(* IEC 61131-3 sources: crb-codesys/generation/scripts/repoeval/重型运输系统/core/PRG, 12 files *)

(* ---- Barrier.st ---- *)
PROGRAM Barrier
VAR
	bInit			:BOOL:=TRUE;
	initCount		:INT:= 100 * 2;		//2s后开始初始化，执行
	timeout			:INT:= 100 * 16;	//10ms间隔时 is 15 second
	timeexe			:INT:= 100 * 8;		//需要停止时，额外执行指令时间
	cmdExecutor0	:CommandExecutor0;
	cmdExecutor		:CommandExecutor;
	grdPid			:ARRAY[1..10] OF grdPosCtrl;
	skyPid			:ARRAY[0..10] OF skyPosCtrl;
	resetPidParam	:BOOL;							//pid参数复位
	pidMode			:BOOL;							//使用pid控制
	autoButtonMode	:BOOL;							//手动复位按钮
	autoEnableMode	:BOOL;							//有动作时使能自动开启
	autoPctMode		:BOOL;
	manualPidPrmSet	:BOOL;							//manualPidParamSet,手动设定pid位置参数

	gi				:INT;			//ground-i
	si				:INT;			//sky-i

	level			:INT;			//1->地轨	2->天轨
	idx				:INT := -1 ;	//挡板索引编号
END_VAR

//初始化
IF initCount = 0 THEN
	IF bInit THEN
		initialize();
		initializePid();
		bInit := FALSE;
	END_IF
ELSE
	initCount := initCount - 1;
	RETURN;
END_IF

//指令执行
pidTestUi();

IF pidMode THEN
	pidCalc();
	pidExecute();
ELSE
	IF autoPctMode THEN setExecutePercent(); END_IF
	manualExecute();
END_IF

//界面交互
interfaceAct();

//状态更新
updateStatus(error := 1);

//复位按钮模式/
IF autoButtonMode THEN
	autoResetButton();
END_IF
IF autoEnableMode THEN
	autoEnable();
END_IF

(* ---- Barrier_autoEnable.st ---- *)
IF pidMode THEN 	//pid模式，没有动作指令时不执行输出

	IF NOT manualPidPrmSet THEN
		FOR gi := 1 TO 10 DO
			 IF gDev.grd[gi].vector = TargetDirect.stop THEN
				cmdExecutor(level := 1, idx := gi, percent := 0);
			 END_IF
		END_FOR

		FOR si := 1 TO 10 DO
			IF gDev.sky[si].vector = TargetDirect.stop THEN
				cmdExecutor(level := 2, idx := si, percent := 0);
			END_IF
		END_FOR
		//起竖挡板执行开关量特判
		IF gDev.sky[0].vector = TargetDirect.stop THEN
			cmdExecutor(level := 2, idx := 0, percent := 0);
		END_IF
	END_IF
ELSE		//开关量控制

	FOR gi := 1 TO 10 DO
		 IF gDev.grd[gi].vector = TargetDirect.stop THEN
			gUI.grd[gi].pwrEnable := FALSE;
		 ELSE
			gUI.grd[gi].pwrEnable := TRUE;
		 END_IF
	END_FOR

	FOR si := 0 TO 10 DO
		IF gDev.sky[si].vector = TargetDirect.stop THEN
			gUI.sky[si].pwrEnable := FALSE;
		ELSE
			gUI.sky[si].pwrEnable := TRUE;
		END_IF
	END_FOR
END_IF

(*
FOR gi := 1 TO 10 DO
	 IF gDev.grd[gi].vector <> TargetDirect.stop THEN
		IF pidMode THEN
			cmdExecutor(level := 1, idx := gi, percent := grdPid[gi].res);
		ELSE
			gUI.grd[gi].pwrEnable := TRUE;
		END_IF
	 ELSE
		IF pidMode THEN
			cmdExecutor(level := 1, idx := gi, percent := 0);
		ELSE
			gUI.grd[gi].pwrEnable := FALSE;
		END_IF
	 END_IF
END_FOR

FOR si := 1 TO 10 DO
	IF gDev.sky[si].vector <> TargetDirect.stop THEN		//运动状态，执行  PID或开关使能
		IF pidMode THEN
			cmdExecutor(level := 2, idx := si, percent := skyPid[si].res);
		ELSE
			gUI.sky[si].pwrEnable := TRUE;
		END_IF
	ELSE													//停止状态，关闭 PID或开关使能
		IF pidMode THEN
			cmdExecutor(level := 2, idx := si, percent := 0);
		ELSE
			gUI.sky[si].pwrEnable := FALSE;
		END_IF
	END_IF
END_FOR

IF gDev.sky[0].vector <> TargetDirect.stop THEN
	gUI.sky[0].pwrEnable := TRUE;
	IF gDev.sky[0].vector = TargetDirect.extend THEN	cmdExecutor(level := 2, idx := 0, percent := gDev.sky[0].ctrl.exPct);END_IF
	IF gDev.sky[0].vector = TargetDirect.retract THEN	cmdExecutor(level := 2, idx := 0, percent := -gDev.sky[0].ctrl.rtPct);END_IF
ELSE
	gUI.sky[0].pwrEnable := FALSE;
	cmdExecutor(level := 2, idx := 0, percent := 0);
END_IF
*)

(* ---- Barrier_autoReseButton.st ---- *)
//更新Button
FOR gi := 1 TO 10 DO
	setButtonByDirect(1, gi, gDev.grd[gi].vector);
END_FOR

FOR si := 0 TO 10 DO
	setButtonByDirect(2, si, gDev.sky[si].vector);
END_FOR

(* ---- Barrier_initialize.st ---- *)
//默认自动使能
gUI.mode.autoEnable	:= TRUE;
gUI.mode.usePID := TRUE;

//initialize boundary val
	//ground
	gDev.grd[	1	].sensor.retractVal	:=	4.4	;		gDev.grd[	1	].sensor.extendVal	:=	108 	;
	gDev.grd[	2	].sensor.retractVal	:=	3.5	;		gDev.grd[	2	].sensor.extendVal	:=	113.4	;
	gDev.grd[	3	].sensor.retractVal	:=	4.1	;		gDev.grd[	3	].sensor.extendVal	:=	110 	;
	gDev.grd[	4	].sensor.retractVal	:=	1	;		gDev.grd[	4	].sensor.extendVal	:=	112.3	;		//结构问题暂不动
	gDev.grd[	5	].sensor.retractVal	:=	4.0	;		gDev.grd[	5	].sensor.extendVal	:=	107.1-0.5	;
	gDev.grd[	6	].sensor.retractVal	:=	3.5	;		gDev.grd[	6	].sensor.extendVal	:=	110.5	;
	gDev.grd[	7	].sensor.retractVal	:=	5	;		gDev.grd[	7	].sensor.extendVal	:=	109.7   ;
	gDev.grd[	8	].sensor.retractVal	:=	4.8	;		gDev.grd[	8	].sensor.extendVal	:=	109.2	;
	gDev.grd[	9	].sensor.retractVal	:=	3.2	;		gDev.grd[	9	].sensor.extendVal	:=	108 -0.5 	;
	gDev.grd[	10	].sensor.retractVal	:=	6.9	;		gDev.grd[	10	].sensor.extendVal	:=	112 	;
(*
	gDev.grd[	7	].sensor.retractVal	:=	3.6	;		gDev.grd[	7	].sensor.extendVal	:=	108.3	;
	gDev.grd[	8	].sensor.retractVal	:=	3.5	;		gDev.grd[	8	].sensor.extendVal	:=	113.1	;
	gDev.grd[	9	].sensor.retractVal	:=	3.2	;		gDev.grd[	9	].sensor.extendVal	:=	107.3	;
	gDev.grd[	10	].sensor.retractVal	:=	3.4	;		gDev.grd[	10	].sensor.extendVal	:=	113.5	;*)

	//sky
	gDev.sky[	0	].sensor.retractVal	:=	3.7	;		gDev.sky[	0	].sensor.extendVal	:=	213.6	;
	gDev.sky[	1	].sensor.retractVal	:=	8.8	;		gDev.sky[	1	].sensor.extendVal	:=	113.1	;
	gDev.sky[	2	].sensor.retractVal	:=	3.5	;		gDev.sky[	2	].sensor.extendVal	:=	113.0	;
	gDev.sky[	3	].sensor.retractVal	:=	3.5	;		gDev.sky[	3	].sensor.extendVal	:=	111.0	;
	gDev.sky[	4	].sensor.retractVal	:=	1	;		gDev.sky[	4	].sensor.extendVal	:=	58.2	;
	gDev.sky[	5	].sensor.retractVal	:=	3.2	;		gDev.sky[	5	].sensor.extendVal	:=	106.6	;
	gDev.sky[	6	].sensor.retractVal	:=	6.2	;		gDev.sky[	6	].sensor.extendVal	:=	109.8	;
(*
	gDev.sky[	7	].sensor.retractVal	:=	1	;		gDev.sky[	7	].sensor.extendVal	:=	113.4	;		//default:115
	gDev.sky[	8	].sensor.retractVal	:=	1	;		gDev.sky[	8	].sensor.extendVal	:=	112.2	;
	gDev.sky[	9	].sensor.retractVal	:=	1	;		gDev.sky[	9	].sensor.extendVal	:=	112.3	;
	gDev.sky[	10	].sensor.retractVal	:=	1	;		gDev.sky[	10	].sensor.extendVal	:=	66.3	;
*)

	gDev.sky[	7	].sensor.retractVal	:=	5	;		gDev.sky[	7	].sensor.extendVal	:=	108.7	;		//default:115
	gDev.sky[	8	].sensor.retractVal	:=	8.6	;		gDev.sky[	8	].sensor.extendVal	:=	113.3	;
	gDev.sky[	9	].sensor.retractVal	:=	12.9 ;		gDev.sky[	9	].sensor.extendVal	:=	113.8	;
	gDev.sky[	10	].sensor.retractVal	:=	3.9 ;		gDev.sky[	10	].sensor.extendVal	:=	111.5	;

//初始化默认伸缩比例量
	gDev.grd[1].ctrl.exPct :=	28		;			gDev.grd[1].ctrl.rtPct :=	25		;
	gDev.grd[2].ctrl.exPct :=	28		;			gDev.grd[2].ctrl.rtPct :=	25		;
	gDev.grd[3].ctrl.exPct :=	30		;			gDev.grd[3].ctrl.rtPct :=	25		;
	gDev.grd[4].ctrl.exPct :=	28		;			gDev.grd[4].ctrl.rtPct :=	25		;
	gDev.grd[5].ctrl.exPct :=	33		;			gDev.grd[5].ctrl.rtPct :=	33		;		//exPct:=26	rtPct:=21 二次比例
	gDev.grd[6].ctrl.exPct :=	28		;			gDev.grd[6].ctrl.rtPct :=	25		;
	gDev.grd[7].ctrl.exPct :=	28		;			gDev.grd[7].ctrl.rtPct :=	25		;
	gDev.grd[8].ctrl.exPct :=	28		;			gDev.grd[8].ctrl.rtPct :=	25		;
	gDev.grd[9].ctrl.exPct :=	28		;			gDev.grd[9].ctrl.rtPct :=	25		;
	gDev.grd[10].ctrl.exPct :=	28		;			gDev.grd[10].ctrl.rtPct :=	25		;

	gDev.sky[0].ctrl.exPct :=	35		;			gDev.sky[0].ctrl.rtPct :=	41		;
	gDev.sky[1].ctrl.exPct :=	25		;			gDev.sky[1].ctrl.rtPct :=	28		;
	gDev.sky[2].ctrl.exPct :=	25		;			gDev.sky[2].ctrl.rtPct :=	28		;
	gDev.sky[3].ctrl.exPct :=	25		;			gDev.sky[3].ctrl.rtPct :=	28		;
	gDev.sky[4].ctrl.exPct :=	25		;			gDev.sky[4].ctrl.rtPct :=	28		;
	gDev.sky[5].ctrl.exPct :=	27		;			gDev.sky[5].ctrl.rtPct :=	30.5	;
	gDev.sky[6].ctrl.exPct :=	25		;			gDev.sky[6].ctrl.rtPct :=	29		;
	gDev.sky[7].ctrl.exPct :=	25		;			gDev.sky[7].ctrl.rtPct :=	28		;
	gDev.sky[8].ctrl.exPct :=	25		;			gDev.sky[8].ctrl.rtPct :=	28		;
	gDev.sky[9].ctrl.exPct :=	25		;			gDev.sky[9].ctrl.rtPct :=	28		;
	gDev.sky[10].ctrl.exPct :=	25		;			gDev.sky[10].ctrl.rtPct :=	28		;

//initialize device name

											gUI.sky[	0	].wname	:=	"天轨1#"	;
gUI.grd[	1	].wname	:=	"地轨1#"	;	gUI.sky[	1	].wname	:=	"天轨2#"	;
gUI.grd[	2	].wname	:=	"地轨2#"	;	gUI.sky[	2	].wname	:=	"天轨3#"	;
gUI.grd[	3	].wname	:=	"地轨3#"	;	gUI.sky[	3	].wname	:=	"天轨4#"	;
gUI.grd[	4	].wname	:=	"地轨4#"	;	gUI.sky[	4	].wname	:=	"天轨5#"	;
gUI.grd[	5	].wname	:=	"地轨5#"	;	gUI.sky[	5	].wname	:=	"天轨6#"	;
gUI.grd[	6	].wname	:=	"地轨6#"	;	gUI.sky[	6	].wname	:=	"天轨7#"	;
gUI.grd[	7	].wname	:=	"地轨7#"	;	gUI.sky[	7	].wname	:=	"天轨8#"	;
gUI.grd[	8	].wname	:=	"地轨8#"	;	gUI.sky[	8	].wname	:=	"天轨9#"	;
gUI.grd[	9	].wname	:=	"地轨9#"	;	gUI.sky[	9	].wname	:=	"天轨10#"	;
gUI.grd[	10	].wname	:=	"地轨10#"	;	gUI.sky[	10	].wname	:=	"天轨11#"	;

												gUI.sky[	0	].hzname	:=	"天.起竖"	;
gUI.grd[	1	].hzname	:=	"地.横1"	;	gUI.sky[	1	].hzname	:=	"天.横1"	;
gUI.grd[	2	].hzname	:=	"地.纵1"	;	gUI.sky[	2	].hzname	:=	"天.纵1"	;
gUI.grd[	3	].hzname	:=	"地.横2"	;	gUI.sky[	3	].hzname	:=	"天.横2"	;
gUI.grd[	4	].hzname	:=	"地.横3"	;	gUI.sky[	4	].hzname	:=	"天.横3"	;
gUI.grd[	5	].hzname	:=	"地.横4"	;	gUI.sky[	5	].hzname	:=	"天.横4"	;
gUI.grd[	6	].hzname	:=	"地.横5"	;	gUI.sky[	6	].hzname	:=	"天.横5"	;
gUI.grd[	7	].hzname	:=	"地.纵2"	;	gUI.sky[	7	].hzname	:=	"天.纵2"	;
gUI.grd[	8	].hzname	:=	"地.横6"	;	gUI.sky[	8	].hzname	:=	"天.横6"	;
gUI.grd[	9	].hzname	:=	"地.横7"	;	gUI.sky[	9	].hzname	:=	"天.横7"	;
gUI.grd[	10	].hzname	:=	"地.横8"	;	gUI.sky[	10	].hzname	:=	"天.横8"	;

											gUI.sky[	0	].name	:=	'SKY_00'	;
gUI.grd[	1	].name	:=	'GRD_01'	;	gUI.sky[	1	].name	:=	'SKY_01'	;
gUI.grd[	2	].name	:=	'GRD_02'	;	gUI.sky[	2	].name	:=	'SKY_02'	;
gUI.grd[	3	].name	:=	'GRD_03'	;	gUI.sky[	3	].name	:=	'SKY_03'	;
gUI.grd[	4	].name	:=	'GRD_04'	;	gUI.sky[	4	].name	:=	'SKY_04'	;
gUI.grd[	5	].name	:=	'GRD_05'	;	gUI.sky[	5	].name	:=	'SKY_05'	;
gUI.grd[	6	].name	:=	'GRD_06'	;	gUI.sky[	6	].name	:=	'SKY_06'	;
gUI.grd[	7	].name	:=	'GRD_07'	;	gUI.sky[	7	].name	:=	'SKY_07'	;
gUI.grd[	8	].name	:=	'GRD_08'	;	gUI.sky[	8	].name	:=	'SKY_08'	;
gUI.grd[	9	].name	:=	'GRD_09'	;	gUI.sky[	9	].name	:=	'SKY_09'	;
gUI.grd[	10	].name	:=	'GRD_10'	;	gUI.sky[	10	].name	:=	'SKY_10'	;

//使用传感器当前位置作为初始化目标位移点
//(*
FOR gi := 1 TO 10 DO
	IF gDev.grd[gi].sensor.position <> 0.0 THEN
		gDev.grd[gi].ctrl.pos.Set_Point := gDev.grd[gi].sensor.position;
	ELSE
		gDev.grd[gi].ctrl.isError := TRUE;
	END_IF
END_FOR

FOR si := 0 TO 10 DO
	IF gDev.sky[si].sensor.position <> 0.0 THEN
		gDev.sky[si].ctrl.pos.Set_Point := gDev.sky[si].sensor.position;
	ELSE
		gDev.sky[si].ctrl.isError := TRUE;
	END_IF
END_FOR
//*)

(* ---- Barrier_initializePid.st ---- *)
//PID param
gDev.grd[	1	].ctrl.pos.Kp	:=	1.2	;	gDev.grd[	1	].ctrl.spd.Kp	:=	0.05	;
gDev.grd[	1	].ctrl.pos.Ki	:=	0	;	gDev.grd[	1	].ctrl.spd.Ki	:=	0		;
gDev.grd[	1	].ctrl.pos.Kd	:=	0	;	gDev.grd[	1	].ctrl.spd.Kd	:=	0.02	;

gDev.grd[	2	].ctrl.pos.Kp	:=	1.3	;	gDev.grd[	2	].ctrl.spd.Kp	:=	0.05	;
gDev.grd[	2	].ctrl.pos.Ki	:=	0	;	gDev.grd[	2	].ctrl.spd.Ki	:=	0		;
gDev.grd[	2	].ctrl.pos.Kd	:=	0	;	gDev.grd[	2	].ctrl.spd.Kd	:=	0.002	;
gDev.grd[	3	].ctrl.pos.Kp	:=	1	;	gDev.grd[	3	].ctrl.spd.Kp	:=	0.01	;
gDev.grd[	3	].ctrl.pos.Ki	:=	0	;	gDev.grd[	3	].ctrl.spd.Ki	:=	0		;
gDev.grd[	3	].ctrl.pos.Kd	:=	0	;	gDev.grd[	3	].ctrl.spd.Kd	:=	0		;

gDev.grd[	4	].ctrl.pos.Kp	:=	0	;	gDev.grd[	4	].ctrl.spd.Kp	:=	0		;
gDev.grd[	4	].ctrl.pos.Ki	:=	0	;	gDev.grd[	4	].ctrl.spd.Ki	:=	0		;
gDev.grd[	4	].ctrl.pos.Kd	:=	0	;	gDev.grd[	4	].ctrl.spd.Kd	:=	0		;
gDev.grd[	5	].ctrl.pos.Kp	:=	1.2	;	gDev.grd[	5	].ctrl.spd.Kp	:=	0.01	;
gDev.grd[	5	].ctrl.pos.Ki	:=	0	;	gDev.grd[	5	].ctrl.spd.Ki	:=	0		;
gDev.grd[	5	].ctrl.pos.Kd	:=	0	;	gDev.grd[	5	].ctrl.spd.Kd	:=	0		;

gDev.grd[	6	].ctrl.pos.Kp	:=	1.2	;	gDev.grd[	6	].ctrl.spd.Kp	:=	0.01	;
gDev.grd[	6	].ctrl.pos.Ki	:=	0	;	gDev.grd[	6	].ctrl.spd.Ki	:=	0		;
gDev.grd[	6	].ctrl.pos.Kd	:=	0	;	gDev.grd[	6	].ctrl.spd.Kd	:=	0		;
gDev.grd[	7	].ctrl.pos.Kp	:=	1.1	;	gDev.grd[	7	].ctrl.spd.Kp	:=	0.02		;
gDev.grd[	7	].ctrl.pos.Ki	:=	0	;	gDev.grd[	7	].ctrl.spd.Ki	:=	0		;
gDev.grd[	7	].ctrl.pos.Kd	:=	0	;	gDev.grd[	7	].ctrl.spd.Kd	:=	0		;

gDev.grd[	8	].ctrl.pos.Kp	:=	1.1	;	gDev.grd[	8	].ctrl.spd.Kp	:=	0.01		;
gDev.grd[	8	].ctrl.pos.Ki	:=	0	;	gDev.grd[	8	].ctrl.spd.Ki	:=	0		;
gDev.grd[	8	].ctrl.pos.Kd	:=	0	;	gDev.grd[	8	].ctrl.spd.Kd	:=	0		;
gDev.grd[	9	].ctrl.pos.Kp	:=	1.1	;	gDev.grd[	9	].ctrl.spd.Kp	:=	0.05		;
gDev.grd[	9	].ctrl.pos.Ki	:=	0	;	gDev.grd[	9	].ctrl.spd.Ki	:=	0		;
gDev.grd[	9	].ctrl.pos.Kd	:=	0	;	gDev.grd[	9	].ctrl.spd.Kd	:=	0		;
gDev.grd[	10	].ctrl.pos.Kp	:=	1.1	;	gDev.grd[	10	].ctrl.spd.Kp	:=	0.02		;
gDev.grd[	10	].ctrl.pos.Ki	:=	0	;	gDev.grd[	10	].ctrl.spd.Ki	:=	0		;
gDev.grd[	10	].ctrl.pos.Kd	:=	0	;	gDev.grd[	10	].ctrl.spd.Kd	:=	0		;

gDev.sky[	0	].ctrl.pos.Kp	:=	1.0	;	gDev.sky[	0	].ctrl.spd.Kp	:=	0.01	;
gDev.sky[	0	].ctrl.pos.Ki	:=	0	;	gDev.sky[	0	].ctrl.spd.Ki	:=	0		;
gDev.sky[	0	].ctrl.pos.Kd	:=	0.1	;	gDev.sky[	0	].ctrl.spd.Kd	:=	0.001	;
gDev.sky[	1	].ctrl.pos.Kp	:=	1.0	;	gDev.sky[	1	].ctrl.spd.Kp	:=	0.01	;
gDev.sky[	1	].ctrl.pos.Ki	:=	0	;	gDev.sky[	1	].ctrl.spd.Ki	:=	0		;
gDev.sky[	1	].ctrl.pos.Kd	:=	0	;	gDev.sky[	1	].ctrl.spd.Kd	:=	0.001	;

gDev.sky[	2	].ctrl.pos.Kp	:=	1.1	;	gDev.sky[	2	].ctrl.spd.Kp	:=	0.02	;
gDev.sky[	2	].ctrl.pos.Ki	:=	0	;	gDev.sky[	2	].ctrl.spd.Ki	:=	0		;
gDev.sky[	2	].ctrl.pos.Kd	:=	0	;	gDev.sky[	2	].ctrl.spd.Kd	:=	0.001	;
gDev.sky[	3	].ctrl.pos.Kp	:=	1.1	;	gDev.sky[	3	].ctrl.spd.Kp	:=	0.02	;
gDev.sky[	3	].ctrl.pos.Ki	:=	0	;	gDev.sky[	3	].ctrl.spd.Ki	:=	0		;
gDev.sky[	3	].ctrl.pos.Kd	:=	0.02;	gDev.sky[	3	].ctrl.spd.Kd	:=	0.001	;

gDev.sky[	4	].ctrl.pos.Kp	:=	0	;	gDev.sky[	4	].ctrl.spd.Kp	:=	0		;
gDev.sky[	4	].ctrl.pos.Ki	:=	0	;	gDev.sky[	4	].ctrl.spd.Ki	:=	0		;
gDev.sky[	4	].ctrl.pos.Kd	:=	0	;	gDev.sky[	4	].ctrl.spd.Kd	:=	0		;
gDev.sky[	5	].ctrl.pos.Kp	:=	1.2	;	gDev.sky[	5	].ctrl.spd.Kp	:=	0.01	;
gDev.sky[	5	].ctrl.pos.Ki	:=	0	;	gDev.sky[	5	].ctrl.spd.Ki	:=	0		;
gDev.sky[	5	].ctrl.pos.Kd	:=	0	;	gDev.sky[	5	].ctrl.spd.Kd	:=	0.001	;

gDev.sky[	6	].ctrl.pos.Kp	:=	1.1	;	gDev.sky[	6	].ctrl.spd.Kp	:=	0.01	;
gDev.sky[	6	].ctrl.pos.Ki	:=	0	;	gDev.sky[	6	].ctrl.spd.Ki	:=	0		;
gDev.sky[	6	].ctrl.pos.Kd	:=	0.01;	gDev.sky[	6	].ctrl.spd.Kd	:=	0.001	;
gDev.sky[	7	].ctrl.pos.Kp	:=	1.1	;	gDev.sky[	7	].ctrl.spd.Kp	:=	0.01	;
gDev.sky[	7	].ctrl.pos.Ki	:=	0	;	gDev.sky[	7	].ctrl.spd.Ki	:=	0		;
gDev.sky[	7	].ctrl.pos.Kd	:=	0	;	gDev.sky[	7	].ctrl.spd.Kd	:=	0		;

gDev.sky[	8	].ctrl.pos.Kp	:=	1.1	;	gDev.sky[	8	].ctrl.spd.Kp	:=	0.01	;
gDev.sky[	8	].ctrl.pos.Ki	:=	0	;	gDev.sky[	8	].ctrl.spd.Ki	:=	0		;
gDev.sky[	8	].ctrl.pos.Kd	:=	0	;	gDev.sky[	8	].ctrl.spd.Kd	:=	0		;
gDev.sky[	9	].ctrl.pos.Kp	:=	1.2	;	gDev.sky[	9	].ctrl.spd.Kp	:=	0.01		;
gDev.sky[	9	].ctrl.pos.Ki	:=	0	;	gDev.sky[	9	].ctrl.spd.Ki	:=	0		;
gDev.sky[	9	].ctrl.pos.Kd	:=	0	;	gDev.sky[	9	].ctrl.spd.Kd	:=	0		;
gDev.sky[	10	].ctrl.pos.Kp	:=	1.1	;	gDev.sky[	10	].ctrl.spd.Kp	:=	0		;
gDev.sky[	10	].ctrl.pos.Ki	:=	0	;	gDev.sky[	10	].ctrl.spd.Ki	:=	0		;
gDev.sky[	10	].ctrl.pos.Kd	:=	0	;	gDev.sky[	10	].ctrl.spd.Kd	:=	0		;

gDev.grd[1	].ctrl.ff.pstThreshold	:=	18.5	;	gDev.grd[1	].ctrl.ff.pstKv	:=	0.35 	;
gDev.grd[1	].ctrl.ff.negThreshold	:=	15  	;	gDev.grd[1	].ctrl.ff.negKv	:=	0.27	;
gDev.grd[2	].ctrl.ff.pstThreshold	:=	18  	;	gDev.grd[2	].ctrl.ff.pstKv	:=	0.27	;
gDev.grd[2	].ctrl.ff.negThreshold	:=	16  	;	gDev.grd[2	].ctrl.ff.negKv	:=	0.27	;
gDev.grd[3	].ctrl.ff.pstThreshold	:=	19  	;	gDev.grd[3	].ctrl.ff.pstKv	:=	0.3 	;
gDev.grd[3	].ctrl.ff.negThreshold	:=	16  	;	gDev.grd[3	].ctrl.ff.negKv	:=	0.3 	;
gDev.grd[4	].ctrl.ff.pstThreshold	:=	0   	;	gDev.grd[4	].ctrl.ff.pstKv	:=	0   	;
gDev.grd[4	].ctrl.ff.negThreshold	:=	0   	;	gDev.grd[4	].ctrl.ff.negKv	:=	0   	;
gDev.grd[5	].ctrl.ff.pstThreshold	:=	18  	;	gDev.grd[5	].ctrl.ff.pstKv	:=	0.3 	;
gDev.grd[5	].ctrl.ff.negThreshold	:=	17  	;	gDev.grd[5	].ctrl.ff.negKv	:=	0.3 	;
gDev.grd[6	].ctrl.ff.pstThreshold	:=	18.5	;	gDev.grd[6	].ctrl.ff.pstKv	:=	0.28	;
gDev.grd[6	].ctrl.ff.negThreshold	:=	17  	;	gDev.grd[6	].ctrl.ff.negKv	:=	0.28	;
gDev.grd[7	].ctrl.ff.pstThreshold	:=	17   	;	gDev.grd[7	].ctrl.ff.pstKv	:=	0.36  	;
gDev.grd[7	].ctrl.ff.negThreshold	:=	15   	;	gDev.grd[7	].ctrl.ff.negKv	:=	0.29  	;
gDev.grd[8	].ctrl.ff.pstThreshold	:=	19   	;	gDev.grd[8	].ctrl.ff.pstKv	:=	0.4   	;
gDev.grd[8	].ctrl.ff.negThreshold	:=	17  	;	gDev.grd[8	].ctrl.ff.negKv	:=	0.3   	;
gDev.grd[9	].ctrl.ff.pstThreshold	:=	18   	;	gDev.grd[9	].ctrl.ff.pstKv	:=	0.45   	;
gDev.grd[9	].ctrl.ff.negThreshold	:=	17   	;	gDev.grd[9	].ctrl.ff.negKv	:=	0.28  	;
gDev.grd[10	].ctrl.ff.pstThreshold	:=	19   	;	gDev.grd[10	].ctrl.ff.pstKv	:=	0.30   	;
gDev.grd[10	].ctrl.ff.negThreshold	:=	19.5   	;	gDev.grd[10	].ctrl.ff.negKv	:=	0.25   	;

gDev.sky[0	].ctrl.ff.pstThreshold	:=	22		;	gDev.sky[0	].ctrl.ff.pstKv	:=	0.29	;
gDev.sky[0	].ctrl.ff.negThreshold	:=	18		;	gDev.sky[0	].ctrl.ff.negKv	:=	0.25	;
gDev.sky[1	].ctrl.ff.pstThreshold	:=	14.8	;	gDev.sky[1	].ctrl.ff.pstKv	:=	0.4 	;
gDev.sky[1	].ctrl.ff.negThreshold	:=	18.5	;	gDev.sky[1	].ctrl.ff.negKv	:=	0.32	;
gDev.sky[2	].ctrl.ff.pstThreshold	:=	17.5	;	gDev.sky[2	].ctrl.ff.pstKv	:=	0.33	;
gDev.sky[2	].ctrl.ff.negThreshold	:=	18.3	;	gDev.sky[2	].ctrl.ff.negKv	:=	0.26	;
gDev.sky[3	].ctrl.ff.pstThreshold	:=	17.8	;	gDev.sky[3	].ctrl.ff.pstKv	:=	0.37	;
gDev.sky[3	].ctrl.ff.negThreshold	:=	17.5	;	gDev.sky[3	].ctrl.ff.negKv	:=	0.33	;
gDev.sky[4	].ctrl.ff.pstThreshold	:=	0		;	gDev.sky[4	].ctrl.ff.pstKv	:=	0		;
gDev.sky[4	].ctrl.ff.negThreshold	:=	0		;	gDev.sky[4	].ctrl.ff.negKv	:=	0		;
gDev.sky[5	].ctrl.ff.pstThreshold	:=	18.0	;	gDev.sky[5	].ctrl.ff.pstKv	:=	0.30	;
gDev.sky[5	].ctrl.ff.negThreshold	:=	28.5	;	gDev.sky[5	].ctrl.ff.negKv	:=	0.40	;
gDev.sky[6	].ctrl.ff.pstThreshold	:=	16.8	;	gDev.sky[6	].ctrl.ff.pstKv	:=	0.35	;
gDev.sky[6	].ctrl.ff.negThreshold	:=	18.8	;	gDev.sky[6	].ctrl.ff.negKv	:=	0.29	;
gDev.sky[7	].ctrl.ff.pstThreshold	:=	17.5	;	gDev.sky[7	].ctrl.ff.pstKv	:=	0.32	;
gDev.sky[7	].ctrl.ff.negThreshold	:=	18.5	;	gDev.sky[7	].ctrl.ff.negKv	:=	0.30	;
gDev.sky[8	].ctrl.ff.pstThreshold	:=	18		;	gDev.sky[8	].ctrl.ff.pstKv	:=	0.3		;
gDev.sky[8	].ctrl.ff.negThreshold	:=	20.5	;	gDev.sky[8	].ctrl.ff.negKv	:=	0.25	;
gDev.sky[9	].ctrl.ff.pstThreshold	:=	15.5	;	gDev.sky[9	].ctrl.ff.pstKv	:=	0.38	;
gDev.sky[9	].ctrl.ff.negThreshold	:=	17.0	;	gDev.sky[9	].ctrl.ff.negKv	:=	0.27	;
gDev.sky[10	].ctrl.ff.pstThreshold	:=	17		;	gDev.sky[10	].ctrl.ff.pstKv	:=	0.32	;
gDev.sky[10	].ctrl.ff.negThreshold	:=	17  	;	gDev.sky[10	].ctrl.ff.negKv	:=	0.3		;

//更新pid伸缩设定位置
FOR gi := 1 TO 10 DO
	gDev.grd[gi].ctrl.extVal := gDev.grd[gi].sensor.extendVal;
	gDev.grd[gi].ctrl.rtcVal := gDev.grd[gi].sensor.retractVal;
END_FOR

FOR si := 0 TO 10 DO
	gDev.sky[si].ctrl.extVal := gDev.sky[si].sensor.extendVal;
	gDev.sky[si].ctrl.rtcVal := gDev.sky[si].sensor.retractVal;
END_FOR
//天地轨伸出均可白嫖位移值,缩回动作不行
gDev.grd[1].ctrl.extVal := gDev.grd[1].sensor.extendVal + 4;
gDev.grd[1].ctrl.rtcVal := gDev.grd[1].sensor.retractVal - 5.4;
gDev.grd[2].ctrl.rtcVal := gDev.grd[2].sensor.retractVal - 5.4;
gDev.grd[2].ctrl.extVal := gDev.grd[2].sensor.extendVal + 3;
gDev.grd[3].ctrl.extVal := gDev.grd[3].sensor.extendVal + 6;
gDev.grd[3].ctrl.rtcVal := gDev.grd[3].sensor.retractVal - 10.5;
gDev.grd[5].ctrl.extVal := gDev.grd[5].sensor.extendVal + 2.5;
gDev.grd[5].ctrl.rtcVal := gDev.grd[5].sensor.retractVal - 1.2-2;
gDev.grd[6].ctrl.extVal := gDev.grd[6].sensor.extendVal + 5.5;
gDev.grd[6].ctrl.rtcVal := gDev.grd[6].sensor.retractVal - 5.5;
gDev.grd[7].ctrl.extVal := gDev.grd[7].sensor.extendVal + 5.3;
gDev.grd[7].ctrl.rtcVal := gDev.grd[7].sensor.retractVal - 15;
gDev.grd[8].ctrl.extVal := gDev.grd[8].sensor.extendVal + 7.1;
gDev.grd[8].ctrl.rtcVal := gDev.grd[8].sensor.retractVal - 16.5;
gDev.grd[9].ctrl.extVal := gDev.grd[9].sensor.extendVal + 4  ;
gDev.grd[9].ctrl.rtcVal := gDev.grd[9].sensor.retractVal - 4 ;

gDev.sky[0].ctrl.rtcVal := gDev.sky[0].sensor.retractVal - 9.0;		//2.7
gDev.sky[1].ctrl.extVal := gDev.sky[1].sensor.extendVal + 7;
gDev.sky[1].ctrl.rtcVal := gDev.sky[1].sensor.retractVal - 6.8;
gDev.sky[2].ctrl.extVal := gDev.sky[2].sensor.extendVal + 2;
gDev.sky[2].ctrl.rtcVal := gDev.sky[2].sensor.retractVal - 3.5;
gDev.sky[3].ctrl.extVal := gDev.sky[3].sensor.extendVal + 7.5;
gDev.sky[3].ctrl.rtcVal := gDev.sky[3].sensor.retractVal - 8.5;
gDev.sky[5].ctrl.extVal := gDev.sky[5].sensor.extendVal + 8 ;
gDev.sky[5].ctrl.rtcVal := gDev.sky[5].sensor.retractVal - 13;
gDev.sky[6].ctrl.extVal := gDev.sky[6].sensor.extendVal + 6;
gDev.sky[6].ctrl.rtcVal := gDev.sky[6].sensor.retractVal - 6;
gDev.sky[7].ctrl.extVal := gDev.sky[7].sensor.extendVal + 5;
gDev.sky[7].ctrl.rtcVal := gDev.sky[7].sensor.retractVal - 4.2;
gDev.sky[9].ctrl.extVal := gDev.sky[9].sensor.extendVal + 2.2;
gDev.sky[9].ctrl.rtcVal := gDev.sky[9].sensor.retractVal - 11;
gDev.sky[10].ctrl.extVal := gDev.sky[10].sensor.extendVal + 9;
gDev.sky[10].ctrl.rtcVal := gDev.sky[10].sensor.retractVal - 11;

FOR gi := 1 TO 10 DO
	gDev.grd[	gi	].ctrl.pos.Max_Val	:=	60	;
	gDev.grd[	gi	].ctrl.pos.Max_ACC	:=	120	;
	gDev.grd[	gi	].ctrl.spd.Max_Val	:=	40	;
	gDev.grd[	gi	].ctrl.spd.Max_ACC	:=	150	;
END_FOR

FOR si := 0 TO 10 DO
	gDev.sky[	si	].ctrl.pos.Max_Val	:=	60	;
	gDev.sky[	si	].ctrl.pos.Max_ACC	:=	120	;
	gDev.sky[	si	].ctrl.spd.Max_Val	:=	40	;
	gDev.sky[	si	].ctrl.spd.Max_ACC	:=	150	;
END_FOR

//初始化
IF initCount = 0 THEN
	IF bInit THEN
		initialize();
		initializePid();
		bInit := FALSE;
	END_IF
ELSE
	initCount := initCount - 1;
	RETURN;
END_IF

//指令执行
pidTestUi();

IF pidMode THEN
	pidCalc();
	pidExecute();
ELSE
	IF autoPctMode THEN setExecutePercent(); END_IF
	manualExecute();
END_IF

//界面交互
interfaceAct();

//状态更新
updateStatus(error := 1);

//复位按钮模式/
IF autoButtonMode THEN
	autoResetButton();
END_IF
IF autoEnableMode THEN
	autoEnable();
END_IF

(* ---- Barrier_interfaceAct.st ---- *)
//位移值及伸出百分比参数输出
FOR gi := 1 TO 10 DO
	gUI.grd[gi].postion := gDev.grd[gi].sensor.position;
	gUI.grd[gi].speed := gDev.grd[gi].sensor.speed;
	gUI.grd[gi].extendPercent := percentCalc(1, gi);
END_FOR
FOR si := 0 TO 10 DO
	gUI.sky[si].postion := gDev.sky[si].sensor.position;
	gUI.sky[si].speed := gDev.sky[si].sensor.speed;
	gUI.sky[si].extendPercent := percentCalc(2, si);
END_FOR

//模式判断
pidMode := gUI.mode.usePID;
autoEnableMode := gUI.mode.autoEnable;
autoButtonMode := NOT gUI.mode.manualButtonSet;
autoPctMode := NOT gUI.mode.manualPercentSet;
manualPidPrmSet := gUI.mode.manualSetPid;
//command generetor
FOR gi := 1 TO 10 DO
	IF gUI.grd[gi].btnExtend <> gUI.grd[gi].btnRetract THEN
		gDev.grd[gi].state := DevStatus.runing;
		IF gUI.grd[gi].btnExtend THEN
			gDev.grd[gi].vector := TargetDirect.extend;
			gUI.grd[gi].btnLast := TargetDirect.extend;
		END_IF
		IF gUI.grd[gi].btnRetract THEN
			gDev.grd[gi].vector := TargetDirect.retract;
			gUI.grd[gi].btnLast := TargetDirect.retract;
		END_IF
	ELSE
		IF gUI.grd[gi].btnExtend THEN
			//伸缩指令不能同时发出，检测到后进行动作转换，重置计数器
			gDev.grd[gi].timeCounter := 0;
			gDev.grd[gi].exeCounter := 0;
			IF gUI.grd[gi].btnLast = TargetDirect.retract THEN
				gDev.grd[gi].vector := TargetDirect.extend;
			ELSE
				gDev.grd[gi].vector := TargetDirect.retract;
			END_IF
			setButtonByDirect(1, gi, gDev.grd[gi].vector);
		ELSE
			gDev.grd[gi].vector := TargetDirect.stop;
		END_IF
	END_IF
	IF gUI.grd[gi].btnStop THEN
		gDev.grd[gi].vector := TargetDirect.stop;
		setButtonByDirect(1, gi, gDev.grd[gi].vector);
	END_IF
END_FOR

FOR si := 0 TO 10 DO
	IF gUI.sky[si].btnExtend <> gUI.sky[si].btnRetract THEN
		gDev.sky[si].state := DevStatus.runing;
		IF gUI.sky[si].btnExtend THEN
			gDev.sky[si].vector := TargetDirect.extend;
			gUI.sky[si].btnLast := TargetDirect.extend;
		END_IF
		IF gUI.sky[si].btnRetract THEN
			gDev.sky[si].vector := TargetDirect.retract;
			gUI.sky[si].btnLast := TargetDirect.retract;
		END_IF
	ELSE
		IF gUI.sky[si].btnExtend THEN
			//伸缩指令不能同时发出，检测到后进行动作转换，重置计数器
			gDev.sky[si].timeCounter := 0;
			gDev.sky[si].exeCounter := 0;
			IF gUI.sky[si].btnLast = TargetDirect.retract THEN
				gDev.sky[si].vector := TargetDirect.extend;
			ELSE
				gDev.sky[si].vector := TargetDirect.retract;
			END_IF
			setButtonByDirect(2, si, gDev.sky[si].vector);
		ELSE
			gDev.sky[si].vector := TargetDirect.stop;
		END_IF
	END_IF
	IF gUI.sky[si].btnStop THEN
		gDev.sky[si].vector := TargetDirect.stop;
		setButtonByDirect(1, gi, gDev.grd[gi].vector);
	END_IF
END_FOR

(* ---- Barrier_manualExecute_method.st ---- *)
METHOD manualExecute
VAR_INPUT
END_VAR
VAR
	//targetDirect		:TargetDirect;
END_VAR

FOR gi := 1 TO 10 DO
	IF gUI.grd[gi].pwrEnable THEN
		cmdExecutor0(level := 1, idx := gi,
					direct := gDev.grd[gi].vector,
					percent := gUI.grd[gi].pwrPercent);
	ELSE
		cmdExecutor0(level := 1, idx := gi, direct := 3, percent := 0);
	END_IF
END_FOR

FOR si := 0 TO 10 DO
	IF gUI.sky[si].pwrEnable THEN
		cmdExecutor0(level := 2, idx := si,
					direct := gDev.sky[si].vector,
					percent := gUI.sky[si].pwrPercent);
	ELSE
		cmdExecutor0(level := 2, idx := si, direct := 3, percent := 0);
	END_IF
END_FOR

(* ---- Barrier_pidCalc_method.st ---- *)
METHOD pidCalc
VAR_INPUT
END_VAR
VAR
	vector			:TargetDirect;
END_VAR

FOR gi := 1 TO 10 DO
	IF NOT manualPidPrmSet THEN
		vector := gDev.grd[gi].vector;
		CASE vector OF
			TargetDirect.stop:
			CASE gDev.grd[gi].state OF
				DevStatus.extended:
					gDev.grd[gi].ctrl.pos.Set_Point := gDev.grd[gi].ctrl.extVal;
				DevStatus.retracted:
					gDev.grd[gi].ctrl.pos.Set_Point := gDev.grd[gi].ctrl.rtcVal;
				ELSE
					gDev.grd[gi].ctrl.pos.Set_Point := gDev.grd[gi].sensor.position;
			END_CASE
			TargetDirect.extend:
				gDev.grd[gi].ctrl.pos.Set_Point := gDev.grd[gi].ctrl.extVal;
			TargetDirect.retract:
				gDev.grd[gi].ctrl.pos.Set_Point := gDev.grd[gi].ctrl.rtcVal;
		END_CASE
END_IF

	grdPid[gi](idx := gi, isReset := resetPidParam, cycTimer := 0.01, res => );

END_FOR

FOR si := 0 TO 10 DO
	IF NOT manualPidPrmSet THEN
		vector := gDev.sky[si].vector;
		CASE vector OF
			TargetDirect.stop:
			CASE gDev.sky[si].state OF
				DevStatus.extended:
					gDev.sky[si].ctrl.pos.Set_Point := gDev.sky[si].ctrl.extVal;
				DevStatus.retracted:
					gDev.sky[si].ctrl.pos.Set_Point := gDev.sky[si].ctrl.rtcVal;
				ELSE
					gDev.sky[si].ctrl.pos.Set_Point := gDev.sky[si].sensor.position;
			END_CASE
			TargetDirect.extend:
				gDev.sky[si].ctrl.pos.Set_Point := gDev.sky[si].ctrl.extVal;
			TargetDirect.retract:
				gDev.sky[si].ctrl.pos.Set_Point := gDev.sky[si].ctrl.rtcVal;
		END_CASE

	END_IF
	skyPid[si](idx := si, isReset := resetPidParam, cycTimer := 0.01, res =>);
END_FOR

(* ---- Barrier_pidExecute_method.st ---- *)
METHOD pidExecute
VAR_INPUT
END_VAR
VAR
	vector 		:TargetDirect;
END_VAR

FOR gi := 1 TO 10 DO
	IF gDev.grd[gi].ctrl.isError THEN
		CONTINUE;
	END_IF
	cmdExecutor(level := 1, idx := gi, percent := grdPid[gi].res);
END_FOR

FOR si := 1 TO 10 DO
	IF gDev.sky[si].ctrl.isError THEN
		CONTINUE;
	END_IF
	cmdExecutor(level := 2, idx := si, percent := skyPid[si].res);
END_FOR

//起竖挡板执行开关量
IF NOT gDev.sky[0].ctrl.isError THEN
	IF gDev.sky[0].vector = TargetDirect.extend THEN
		cmdExecutor(level := 2, idx := 0, percent := gDev.sky[0].ctrl.exPct);
	END_IF
	IF gDev.sky[0].vector = TargetDirect.retract THEN
		cmdExecutor(level := 2, idx := 0, percent := -gDev.sky[0].ctrl.rtPct);
	END_IF
END_IF
(*
IF NOT gDev.grd[7].ctrl.isError THEN
	IF gDev.grd[7].vector = TargetDirect.extend THEN
		cmdExecutor(level := 1, idx := 7, percent := gDev.grd[7].ctrl.exPct);
	END_IF
	IF gDev.grd[7].vector = TargetDirect.retract THEN
		cmdExecutor(level := 1, idx := 7, percent := -gDev.grd[7].ctrl.rtPct);
	END_IF
END_IF
IF NOT gDev.sky[7].ctrl.isError THEN
	IF gDev.sky[7].vector = TargetDirect.extend THEN
		cmdExecutor(level := 2, idx := 7, percent := gDev.sky[7].ctrl.exPct);
	END_IF
	IF gDev.sky[7].vector = TargetDirect.retract THEN
		cmdExecutor(level := 2, idx := 7, percent := -gDev.sky[7].ctrl.rtPct);
	END_IF
END_IF
*)

(* ---- Barrier_pidTestUi_method.st ---- *)
METHOD pidTestUi
VAR_INPUT
END_VAR

VAR

END_VAR

IF gUI.pid.level = 1 AND gUI.pid.idx = 0 THEN	//地轨从1-10，天轨从0-10
	RETURN;
END_IF

IF gUI.mode.syncExt THEN
	gUI.grd[gUI.pid.idx].btnExtend := TRUE;gUI.sky[gUI.pid.idx].btnExtend := TRUE;
END_IF
IF gUI.mode.syncRct THEN
	gUI.grd[gUI.pid.idx].btnRetract := TRUE;gUI.sky[gUI.pid.idx].btnRetract := TRUE;
END_IF

IF (NOT gUI.pid.posBtn) THEN
	RETURN;
END_IF

IF gUI.pid.level = 1 THEN 	//地轨部分
	IF idx = gUI.pid.idx THEN		//标号相同更新设备参数

		gUI.pid.devSetPos := gDev.grd[idx].ctrl.pos.Set_Point;
		gUI.pid.executeVal := grdPid[idx].res;
		resetPidParam := gUI.pid.rstPidBtn;
		//-----------------位置环------------------------------//
		gUI.pid.pos.Act_Val := gDev.grd[idx].sensor.position;
		gUI.pid.pos.Err := gUI.pid.pos.Set_Point - gUI.pid.pos.Act_Val;
		gUI.pid.pos.OUT := gDev.grd[idx].ctrl.pos.OUT;
		gDev.grd[idx].ctrl.pos := gUI.pid.pos;
		//-----------------速度环------------------------------//
		gUI.pid.spd.Act_Val := gDev.grd[idx].sensor.speed;
		gUI.pid.spd.Err := gUI.pid.spd.Set_Point - gUI.pid.spd.Act_Val;
		gUI.pid.spd.OUT := gDev.sky[idx].ctrl.spd.OUT;
		gDev.grd[idx].ctrl.spd := gUI.pid.spd;
		//-----------------前馈参数------------------------------//
		gDev.grd[idx].ctrl.ff := gUI.pid.ff;

	ELSE							//标号不同，更新界面参数
		idx := gUI.pid.idx;
		gUI.pid.pos := gDev.grd[idx].ctrl.pos;
		gUI.pid.spd := gDev.grd[idx].ctrl.spd;
		gUI.pid.ff	:= gDev.grd[idx].ctrl.ff;
	END_IF
END_IF
IF gUI.pid.level = 2 THEN 					//天轨部分
	IF idx = gUI.pid.idx THEN		//标号相同更新设备参数

		//-----------------位置环------------------------------//
		gUI.pid.pos.Act_Val := gDev.sky[idx].sensor.position;
		gUI.pid.pos.Err := gUI.pid.pos.Set_Point - gUI.pid.pos.Act_Val;
		gUI.pid.pos.OUT := gDev.sky[idx].ctrl.pos.OUT;
		gDev.sky[idx].ctrl.pos := gUI.pid.pos;
		//-----------------速度环------------------------------//
		gUI.pid.spd.Act_Val := gDev.sky[idx].sensor.speed;
		gUI.pid.spd.Err := gUI.pid.spd.Set_Point - gUI.pid.spd.Act_Val;
		gUI.pid.spd.OUT := gDev.sky[idx].ctrl.spd.OUT;
		gDev.sky[idx].ctrl.spd := gUI.pid.spd;
		//-----------------前馈参数------------------------------//
		gDev.sky[idx].ctrl.ff := gUI.pid.ff;

		gUI.pid.devSetPos := gDev.sky[idx].ctrl.pos.Set_Point;
		gUI.pid.executeVal := skyPid[idx].res;
		resetPidParam := gUI.pid.rstPidBtn;

	ELSE							//标号不同，更新界面参数
		idx := gUI.pid.idx;
		gUI.pid.pos := gDev.sky[idx].ctrl.pos;
		gUI.pid.spd := gDev.sky[idx].ctrl.spd;
		gUI.pid.ff	:= gDev.sky[idx].ctrl.ff;

	END_IF

END_IF

(* ---- Barrier_setExecutePercent.st ---- *)
FOR gi := 1 TO 10 DO
	IF gUI.grd[gi].btnExtend THEN
		gUI.grd[gi].pwrPercent := gDev.grd[gi].ctrl.exPct;
	END_IF
	IF gUI.grd[gi].btnRetract THEN
		gUI.grd[gi].pwrPercent := gDev.grd[gi].ctrl.rtPct;
	END_IF
END_FOR

FOR si := 0 TO 10 DO
	IF gUI.sky[si].btnExtend THEN
		gUI.sky[si].pwrPercent := gDev.sky[si].ctrl.exPct;
	END_IF
	IF gUI.sky[si].btnRetract THEN
		gUI.sky[si].pwrPercent := gDev.sky[si].ctrl.rtPct;
	END_IF
END_FOR

//grd[5]比例输出特判(延时时间过长，小信号无法动作，动作后速度过快的问题)使用速度传感器判定
IF gUI.grd[5].btnExtend THEN
	IF ABS(gDev.grd[5].sensor.extendVal - gDev.grd[5].sensor.position) < 25 THEN
		gUI.grd[5].pwrPercent := 22;
	END_IF
END_IF
IF gUI.grd[5].btnRetract THEN
	IF ABS(gDev.grd[5].sensor.retractVal - gDev.grd[5].sensor.position) < 30 THEN
		gUI.grd[5].pwrPercent := 22;
	END_IF
END_IF

//其他特判
(*IF gUI.grd[2].btnRetract THEN
	IF ABS(gDev.grd[2].sensor.retractVal - gDev.grd[2].sensor.position) < 20 THEN
		gUI.grd[2].pwrPercent := 21;
	END_IFa
END_IF*)
IF gUI.grd[6].btnRetract THEN
	IF ABS(gDev.grd[6].sensor.retractVal - gDev.grd[6].sensor.position) < 25 THEN
		gUI.grd[6].pwrPercent := 21;
	END_IF
END_IF

(* ---- Barrier_updateStatus_method.st ---- *)
METHOD pidTestUi
VAR_INPUT
END_VAR

VAR

END_VAR

IF gUI.pid.level = 1 AND gUI.pid.idx = 0 THEN	//地轨从1-10，天轨从0-10
	RETURN;
END_IF

IF gUI.mode.syncExt THEN
	gUI.grd[gUI.pid.idx].btnExtend := TRUE;gUI.sky[gUI.pid.idx].btnExtend := TRUE;
END_IF
IF gUI.mode.syncRct THEN
	gUI.grd[gUI.pid.idx].btnRetract := TRUE;gUI.sky[gUI.pid.idx].btnRetract := TRUE;
END_IF

IF (NOT gUI.pid.posBtn) THEN
	RETURN;
END_IF

IF gUI.pid.level = 1 THEN 	//地轨部分
	IF idx = gUI.pid.idx THEN		//标号相同更新设备参数

		gUI.pid.devSetPos := gDev.grd[idx].ctrl.pos.Set_Point;
		gUI.pid.executeVal := grdPid[idx].res;
		resetPidParam := gUI.pid.rstPidBtn;
		//-----------------位置环------------------------------//
		gUI.pid.pos.Act_Val := gDev.grd[idx].sensor.position;
		gUI.pid.pos.Err := gUI.pid.pos.Set_Point - gUI.pid.pos.Act_Val;
		gUI.pid.pos.OUT := gDev.grd[idx].ctrl.pos.OUT;
		gDev.grd[idx].ctrl.pos := gUI.pid.pos;
		//-----------------速度环------------------------------//
		gUI.pid.spd.Act_Val := gDev.grd[idx].sensor.speed;
		gUI.pid.spd.Err := gUI.pid.spd.Set_Point - gUI.pid.spd.Act_Val;
		gUI.pid.spd.OUT := gDev.sky[idx].ctrl.spd.OUT;
		gDev.grd[idx].ctrl.spd := gUI.pid.spd;
		//-----------------前馈参数------------------------------//
		gDev.grd[idx].ctrl.ff := gUI.pid.ff;

	ELSE							//标号不同，更新界面参数
		idx := gUI.pid.idx;
		gUI.pid.pos := gDev.grd[idx].ctrl.pos;
		gUI.pid.spd := gDev.grd[idx].ctrl.spd;
		gUI.pid.ff	:= gDev.grd[idx].ctrl.ff;
	END_IF
END_IF
IF gUI.pid.level = 2 THEN 					//天轨部分
	IF idx = gUI.pid.idx THEN		//标号相同更新设备参数

		//-----------------位置环------------------------------//
		gUI.pid.pos.Act_Val := gDev.sky[idx].sensor.position;
		gUI.pid.pos.Err := gUI.pid.pos.Set_Point - gUI.pid.pos.Act_Val;
		gUI.pid.pos.OUT := gDev.sky[idx].ctrl.pos.OUT;
		gDev.sky[idx].ctrl.pos := gUI.pid.pos;
		//-----------------速度环------------------------------//
		gUI.pid.spd.Act_Val := gDev.sky[idx].sensor.speed;
		gUI.pid.spd.Err := gUI.pid.spd.Set_Point - gUI.pid.spd.Act_Val;
		gUI.pid.spd.OUT := gDev.sky[idx].ctrl.spd.OUT;
		gDev.sky[idx].ctrl.spd := gUI.pid.spd;
		//-----------------前馈参数------------------------------//
		gDev.sky[idx].ctrl.ff := gUI.pid.ff;

		gUI.pid.devSetPos := gDev.sky[idx].ctrl.pos.Set_Point;
		gUI.pid.executeVal := skyPid[idx].res;
		resetPidParam := gUI.pid.rstPidBtn;

	ELSE							//标号不同，更新界面参数
		idx := gUI.pid.idx;
		gUI.pid.pos := gDev.sky[idx].ctrl.pos;
		gUI.pid.spd := gDev.sky[idx].ctrl.spd;
		gUI.pid.ff	:= gDev.sky[idx].ctrl.ff;

	END_IF

END_IF
